# B&R Automation Studio project Prog_4
Automation Studio 4.5.2.102

## Configuration Config1

### Task classes (Cpu.sw)
```
Cyclic#1:
  Program <- Program.prg
VcDataObjects: Visu <- Visu.dob
Binaries: vcpfpp30, vcmgr, arsvcreg, arialbd, udbdef, vcpdsw, vcalarm, vccdt, vccbmp, vcgclass, Visu01, vctcal, vcshared, TCData, vccbtn, vcfile, Visu02, vcdsint, Visu03, vcrt, vcpfmtcx, vcbclass, vcfntttf, vcptelo, vcdsloc, vccovl, vcpdpp30, arial, Role, iomap, arconfig, asfw, sysconf, User, ashwac, ashwd
Libraries: McBase, runtime, fileio, vcresman, dataobj
```

### Hardware
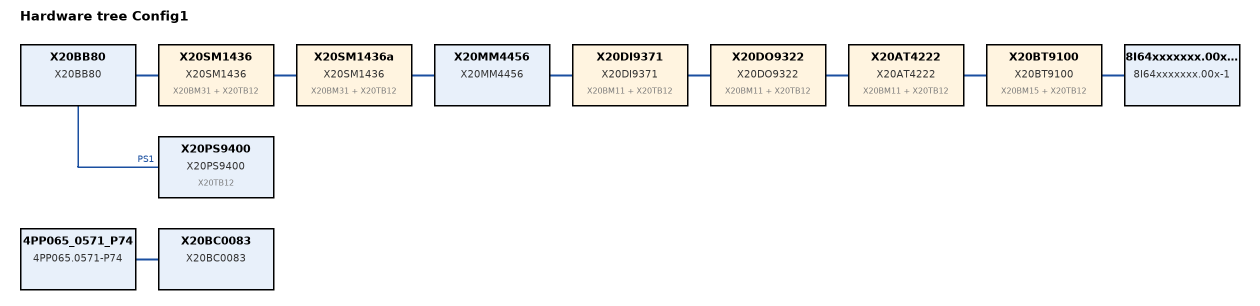
```
4PP065_0571_P74 : 4PP065.0571-P74 v1.1.2.0
  Connector IF5:
    ActivateDevice = 1
    Mode = Manual
    InternetAddress = 10.0.1.10
    SubnetMask = 255.255.255.0
  ConfigurationID = labBR
  VcObjectName = Visu
8I64xxxxxxx.00x-1 : 8I64xxxxxxx.00x-1 v2.1.3.0  [X2X1 -> X20BT9100.X2X1 [Cable Type=X2XCable, Length=10, Version=1.0.0.2]]
  FunctionModel = Standard
  packedETAD = packed
  packedCMDD = packed
X20AT4222 : X20AT4222 v1.2.3.0  [SS1 -> X20TB12c.SS; SL -> X20BM11b.SL1]
X20BB80 : X20BB80 v1.0.2.0
X20BC0083 : X20BC0083 v2.9.0.0  [PLK1 -> 4PP065_0571_P74.IF4 (NodeNumber=2) [Cable Type=PowerlinkCable, Length=10, Version=1.0.0.2]; SL -> X20BB80.SL1]
X20BM11 : X20BM11 v1.0.0.1  [X2X1 -> X20MM4456.X2X2]
X20BM11a : X20BM11 v1.0.0.1  [X2X1 -> X20BM11.X2X2]
X20BM11b : X20BM11 v1.0.0.1  [X2X1 -> X20BM11a.X2X2]
X20BM15 : X20BM15 v1.0.1.0  [X2X1 -> X20BM11b.X2X2 (NodeNumber=10)]
X20BM31 : X20BM31 v1.0.0.1  [X2X1 -> X20BB80.IF1]
X20BM31a : X20BM31 v1.0.0.1  [X2X1 -> X20BM31.X2X2]
X20BT9100 : X20BT9100 v1.0.3.0  [SS1 -> X20TB12f.SS; SL -> X20BM15.SL1]
X20DI9371 : X20DI9371 v1.0.2.0  [SS1 -> X20TB12.SS; SL -> X20BM11.SL1]
X20DO9322 : X20DO9322 v1.0.3.0  [SS1 -> X20TB12a.SS; SL -> X20BM11a.SL1]
X20MM4456 : X20MM4456 v1.1.5.0  [X2X1 -> X20BM31a.X2X2]
X20PS9400 : X20PS9400 v1.8.0.0  [SS1 -> X20TB12b.SS; PS -> X20BB80.PS1]
X20SM1436 : X20SM1436 v2.2.0.0  [SS1 -> X20TB12d.SS; SL -> X20BM31.SL1]
X20SM1436a : X20SM1436 v2.2.0.0  [SS1 -> X20TB12e.SS; SL -> X20BM31a.SL1]
X20TB12 : X20TB12 v1.0.0.0
X20TB12a : X20TB12 v1.0.0.0
X20TB12b : X20TB12 v1.0.0.0
X20TB12c : X20TB12 v1.0.0.0
X20TB12d : X20TB12 v1.0.0.0
X20TB12e : X20TB12 v1.0.0.0
X20TB12f : X20TB12 v1.0.0.0
```

### IoMap.iom - 4PP065_0571_P74/IoMap.iom
```iecst
VAR_CONFIG
	::real_motor_speed AT %IW."8I64xxxxxxx.00x-1".RFRD_Input;
	::motor_speed AT %QW."8I64xxxxxxx.00x-1".LFRD_Output;
	::LED[0] AT %QX."X20DO9322".DigitalOutput02;
	::LED[1] AT %QX."X20DO9322".DigitalOutput03;
	::LED[2] AT %QX."X20DO9322".DigitalOutput04;
	::LED[3] AT %QX."X20DO9322".DigitalOutput05;
END_VAR
```

## Logical view

### Program Logical/Program

#### Variables.var
```iecst
VAR
	blink_time : ARRAY[0..3] OF USINT;
END_VAR
```

#### Main.c
```c
#include <bur/plctypes.h>

#ifdef _DEFAULT_INCLUDES
#include <AsDefault.h>
#endif

void _INIT ProgramInit(void)
{
	srand(time(0));
}

void _CYCLIC ProgramCyclic(void)
{
	int i;
	if (blink) {
		for (i = 0; i < 4; i++) {
			if (blink_time[i] == 0) {
				LED[i] = !LED[i];
				int r = rand() % 21 + 2;
				blink_time[i] += r;
			}
			blink_time[i]--;
		}
	} else {
		for (i = 0; i < 4; i++) LED[i] = BTN[i];
	}
}

void _EXIT ProgramExit(void)
{

}
```
